TYPE SSIEncoderStatuses :
STRUCT
	///Is the device in a healthy state?
	healthStatus: HealthStatus;
END_STRUCT
END_TYPE

(* stored: Version 1.1.0.1, ProductVersion 3.1.4019.2
   DUT SSIEncoderStatuses: Id {5844f249-1747-48d4-a092-db985eaf1964} *)
